// TwinCAT 3 PLC project Teleruptor_Schakeling
// ProgramVersion: 3.1.4024.0
// libraries:
//   Tc2_Standard, * (Beckhoff Automation GmbH)
//   Tc2_System, * (Beckhoff Automation GmbH)
//   Tc3_Module, * (Beckhoff Automation GmbH)
// project tree:
//   / PlcTask.TcTTO
//   POUs/ MAIN.TcPOU

CONFIGURATION Teleruptor_Schakeling
    RESOURCE PLC ON TwinCAT3
        TASK PlcTask(INTERVAL := T#10ms, PRIORITY := 26);
        PROGRAM MAIN WITH PlcTask : MAIN;
    END_RESOURCE
END_CONFIGURATION

// ---- POUs/MAIN.TcPOU
PROGRAM MAIN
VAR
	
// Events
	EV_1: R_TRIG; // Event 1
	EV_2: R_TRIG; // Event 2
	
// Inputs
	DK_1 AT %I*: BOOL; // Drukknop beneden
	DK_2 AT %I*: BOOL; // Drukknop Boven
	
// Outputs
	LAMP AT %Q*: BOOL; // Lamp in de Hal
	
END_VAR

(*
https://infosys.beckhoff.com/english.php?content=../content/1033/tcplclib_tc2_standard/74391563.html&id=

Teleruptorschakeling (2 regels)

Programmeer de teleruptorschakeling in Structured Tekst. 
Zorg ook hier dat het mogelijk is om te bedienen met meerdere drukknoppen. 
Je zal merken dat dit een veel eenvoudiger programma zal zijn dan in LADDER. 

Voor de flank-detectie heb je een Function Block (FB) nodig.
Met een rechtermuisklik in het programmeervenster (niet het declareer venster) kan 
de 'input assisant' openen en selecteer vervolgens > Function Blocks > Tc2_Standard > trigger > R_TRIG
*)


EV_1(CLK:=DK_1 , Q=>LAMP ); 
EV_2(CLK:=DK_2 , Q=>LAMP );

END_PROGRAM
